Fanuc KAREL source: ko00012.KL

-- PROVISIONAL review KL for V1013-1; original PC SHA256 223ebba528226c7bf7cd511b29e175afb0da2dbf77bedb1037b7415ce0c3ce69
-- Incomplete behavior may be omitted. Consult companion uncertainty JSON. Do not deploy.
PROGRAM KO00012
%NOLOCKGROUP
-- UNRESOLVED_DECL P1 type=000102
-- UNRESOLVED_DECL P2 type=000102
-- UNRESOLVED_DECL P3 type=000102
-- UNRESOLVED_DECL OUT type=000199
BEGIN
  -- UNRESOLVED_PC offsets 5-65; opcodes 27,27,49,7E,AD,27,49,7E,AD,27,49,7E,AD,76,7E,4A
  -- UNRESOLVED_PC offsets 70-74; opcodes 7F
END KO00012
